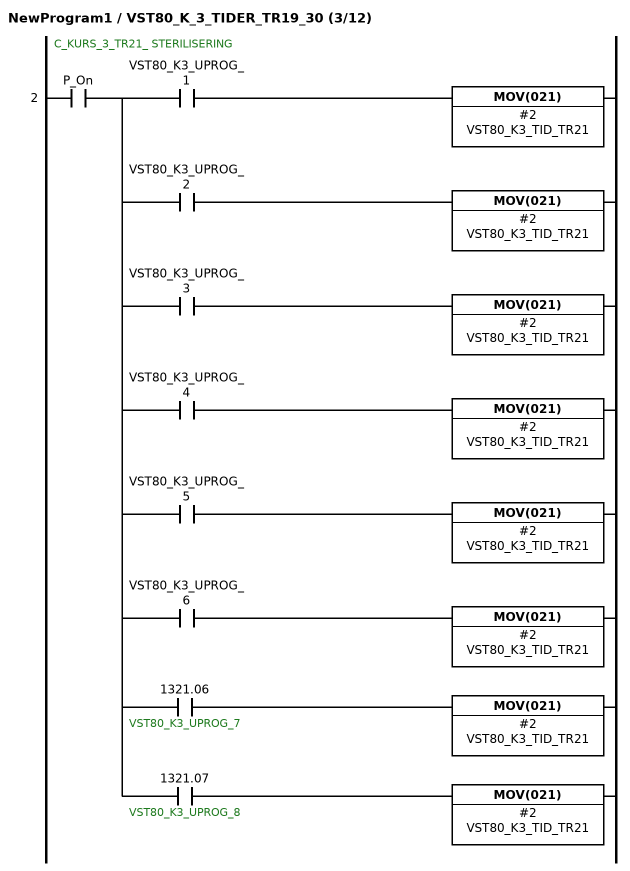
; [picture p312: NewProgram1 / VST80_K_3_TIDER_TR19_30, rungs 2-2]
; rung 2: C_KURS_3_TR21_ STERILISERING
LD P_On
OUT TR0
AND VST80_K3_UPROG_1
MOV(021) #2 VST80_K3_TID_TR21
LD TR0
AND VST80_K3_UPROG_2
MOV(021) #2 VST80_K3_TID_TR21
LD TR0
AND VST80_K3_UPROG_3
MOV(021) #2 VST80_K3_TID_TR21
LD TR0
AND VST80_K3_UPROG_4
MOV(021) #2 VST80_K3_TID_TR21
LD TR0
AND VST80_K3_UPROG_5
MOV(021) #2 VST80_K3_TID_TR21
LD TR0
AND VST80_K3_UPROG_6
MOV(021) #2 VST80_K3_TID_TR21
LD TR0
AND 1321.06  ; VST80_K3_UPROG_7
MOV(021) #2 VST80_K3_TID_TR21
LD TR0
AND 1321.07  ; VST80_K3_UPROG_8
MOV(021) #2 VST80_K3_TID_TR21

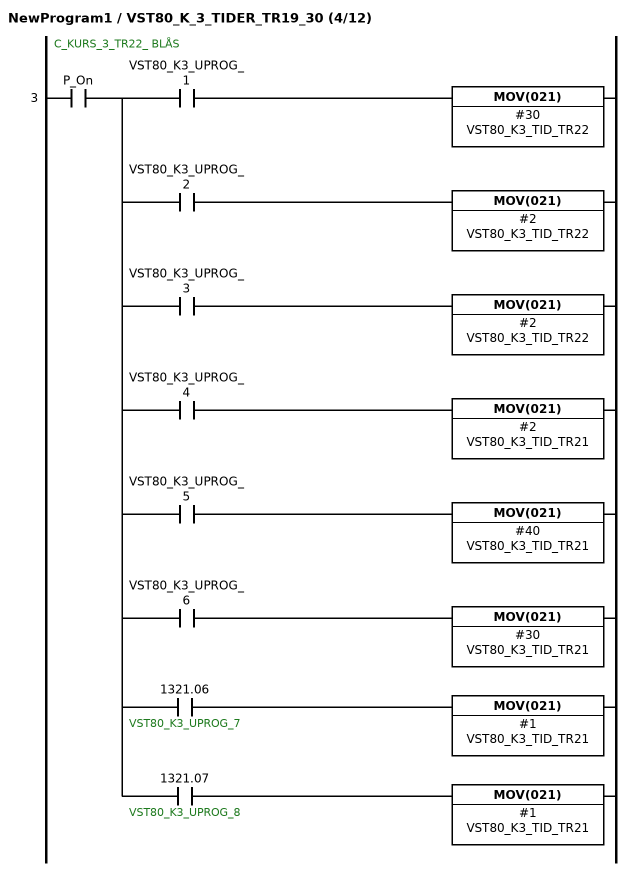
; rung 3: C_KURS_3_TR22_ BLÅS
LD P_On
OUT TR0
AND VST80_K3_UPROG_1
MOV(021) #30 VST80_K3_TID_TR22
LD TR0
AND VST80_K3_UPROG_2
MOV(021) #2 VST80_K3_TID_TR22
LD TR0
AND VST80_K3_UPROG_3
MOV(021) #2 VST80_K3_TID_TR22
LD TR0
AND VST80_K3_UPROG_4
MOV(021) #2 VST80_K3_TID_TR21
LD TR0
AND VST80_K3_UPROG_5
MOV(021) #40 VST80_K3_TID_TR21
LD TR0
AND VST80_K3_UPROG_6
MOV(021) #30 VST80_K3_TID_TR21
LD TR0
AND 1321.06  ; VST80_K3_UPROG_7
MOV(021) #1 VST80_K3_TID_TR21
LD TR0
AND 1321.07  ; VST80_K3_UPROG_8
MOV(021) #1 VST80_K3_TID_TR21

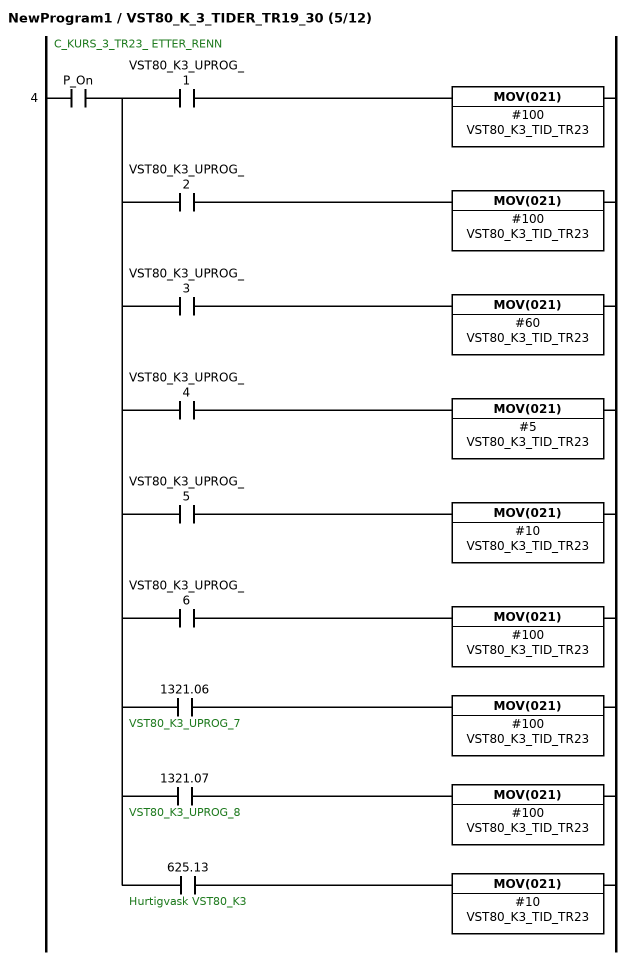
; rung 4: C_KURS_3_TR23_ ETTER_RENN
LD P_On
OUT TR0
AND VST80_K3_UPROG_1
MOV(021) #100 VST80_K3_TID_TR23
LD TR0
AND VST80_K3_UPROG_2
MOV(021) #100 VST80_K3_TID_TR23
LD TR0
AND VST80_K3_UPROG_3
MOV(021) #60 VST80_K3_TID_TR23
LD TR0
AND VST80_K3_UPROG_4
MOV(021) #5 VST80_K3_TID_TR23
LD TR0
AND VST80_K3_UPROG_5
MOV(021) #10 VST80_K3_TID_TR23
LD TR0
AND VST80_K3_UPROG_6
MOV(021) #100 VST80_K3_TID_TR23
LD TR0
AND 1321.06  ; VST80_K3_UPROG_7
MOV(021) #100 VST80_K3_TID_TR23
LD TR0
AND 1321.07  ; VST80_K3_UPROG_8
MOV(021) #100 VST80_K3_TID_TR23
LD TR0
AND 625.13  ; Hurtigvask VST80_K3
MOV(021) #10 VST80_K3_TID_TR23

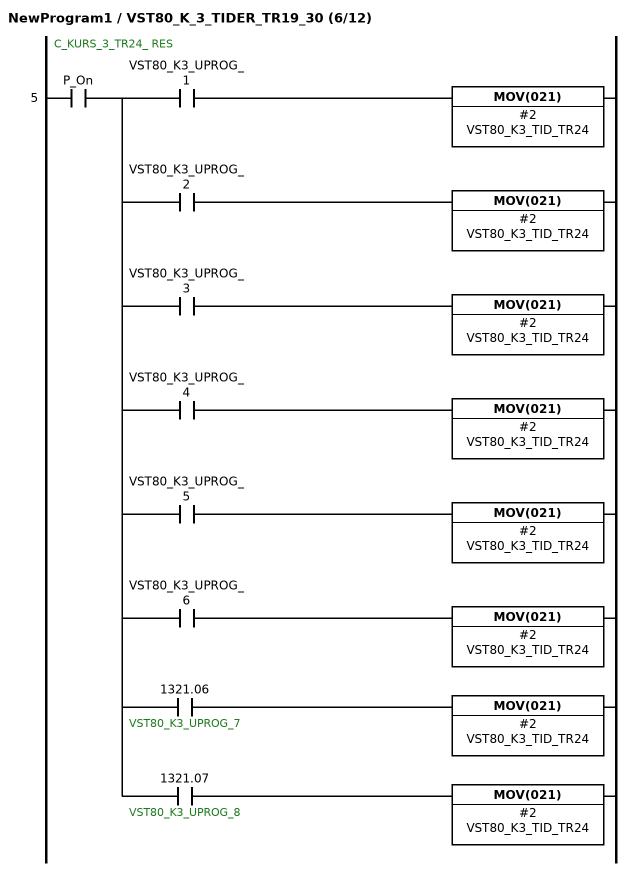
; rung 5: C_KURS_3_TR24_ RES
LD P_On
OUT TR0
AND VST80_K3_UPROG_1
MOV(021) #2 VST80_K3_TID_TR24
LD TR0
AND VST80_K3_UPROG_2
MOV(021) #2 VST80_K3_TID_TR24
LD TR0
AND VST80_K3_UPROG_3
MOV(021) #2 VST80_K3_TID_TR24
LD TR0
AND VST80_K3_UPROG_4
MOV(021) #2 VST80_K3_TID_TR24
LD TR0
AND VST80_K3_UPROG_5
MOV(021) #2 VST80_K3_TID_TR24
LD TR0
AND VST80_K3_UPROG_6
MOV(021) #2 VST80_K3_TID_TR24
LD TR0
AND 1321.06  ; VST80_K3_UPROG_7
MOV(021) #2 VST80_K3_TID_TR24
LD TR0
AND 1321.07  ; VST80_K3_UPROG_8
MOV(021) #2 VST80_K3_TID_TR24

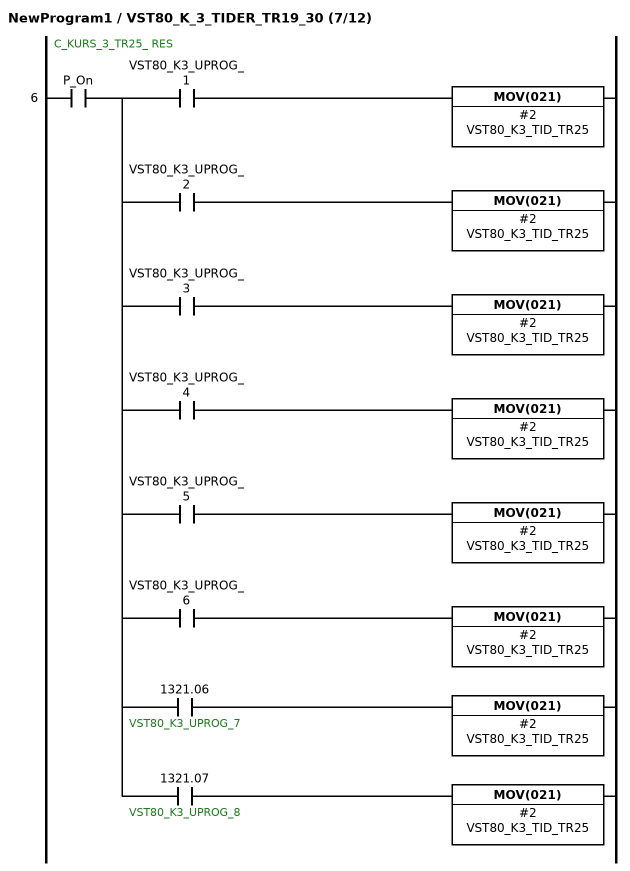
; rung 6: C_KURS_3_TR25_ RES
LD P_On
OUT TR0
AND VST80_K3_UPROG_1
MOV(021) #2 VST80_K3_TID_TR25
LD TR0
AND VST80_K3_UPROG_2
MOV(021) #2 VST80_K3_TID_TR25
LD TR0
AND VST80_K3_UPROG_3
MOV(021) #2 VST80_K3_TID_TR25
LD TR0
AND VST80_K3_UPROG_4
MOV(021) #2 VST80_K3_TID_TR25
LD TR0
AND VST80_K3_UPROG_5
MOV(021) #2 VST80_K3_TID_TR25
LD TR0
AND VST80_K3_UPROG_6
MOV(021) #2 VST80_K3_TID_TR25
LD TR0
AND 1321.06  ; VST80_K3_UPROG_7
MOV(021) #2 VST80_K3_TID_TR25
LD TR0
AND 1321.07  ; VST80_K3_UPROG_8
MOV(021) #2 VST80_K3_TID_TR25

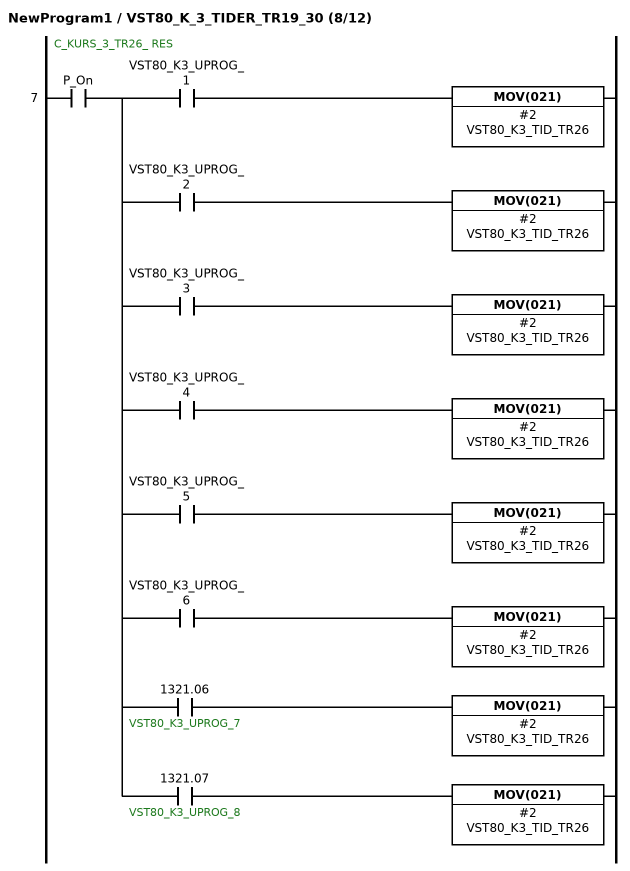
; rung 7: C_KURS_3_TR26_ RES
LD P_On
OUT TR0
AND VST80_K3_UPROG_1
MOV(021) #2 VST80_K3_TID_TR26
LD TR0
AND VST80_K3_UPROG_2
MOV(021) #2 VST80_K3_TID_TR26
LD TR0
AND VST80_K3_UPROG_3
MOV(021) #2 VST80_K3_TID_TR26
LD TR0
AND VST80_K3_UPROG_4
MOV(021) #2 VST80_K3_TID_TR26
LD TR0
AND VST80_K3_UPROG_5
MOV(021) #2 VST80_K3_TID_TR26
LD TR0
AND VST80_K3_UPROG_6
MOV(021) #2 VST80_K3_TID_TR26
LD TR0
AND 1321.06  ; VST80_K3_UPROG_7
MOV(021) #2 VST80_K3_TID_TR26
LD TR0
AND 1321.07  ; VST80_K3_UPROG_8
MOV(021) #2 VST80_K3_TID_TR26

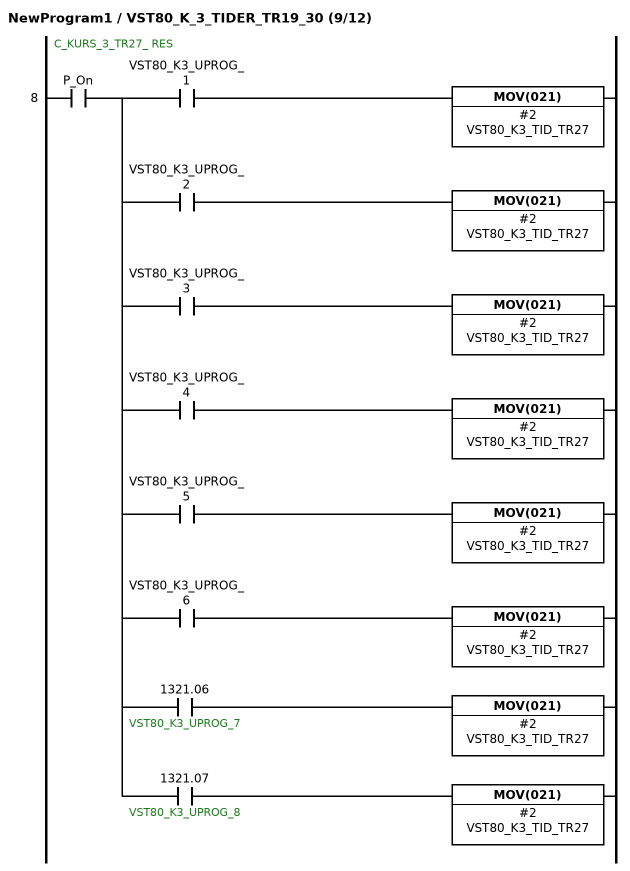
; rung 8: C_KURS_3_TR27_ RES
LD P_On
OUT TR0
AND VST80_K3_UPROG_1
MOV(021) #2 VST80_K3_TID_TR27
LD TR0
AND VST80_K3_UPROG_2
MOV(021) #2 VST80_K3_TID_TR27
LD TR0
AND VST80_K3_UPROG_3
MOV(021) #2 VST80_K3_TID_TR27
LD TR0
AND VST80_K3_UPROG_4
MOV(021) #2 VST80_K3_TID_TR27
LD TR0
AND VST80_K3_UPROG_5
MOV(021) #2 VST80_K3_TID_TR27
LD TR0
AND VST80_K3_UPROG_6
MOV(021) #2 VST80_K3_TID_TR27
LD TR0
AND 1321.06  ; VST80_K3_UPROG_7
MOV(021) #2 VST80_K3_TID_TR27
LD TR0
AND 1321.07  ; VST80_K3_UPROG_8
MOV(021) #2 VST80_K3_TID_TR27

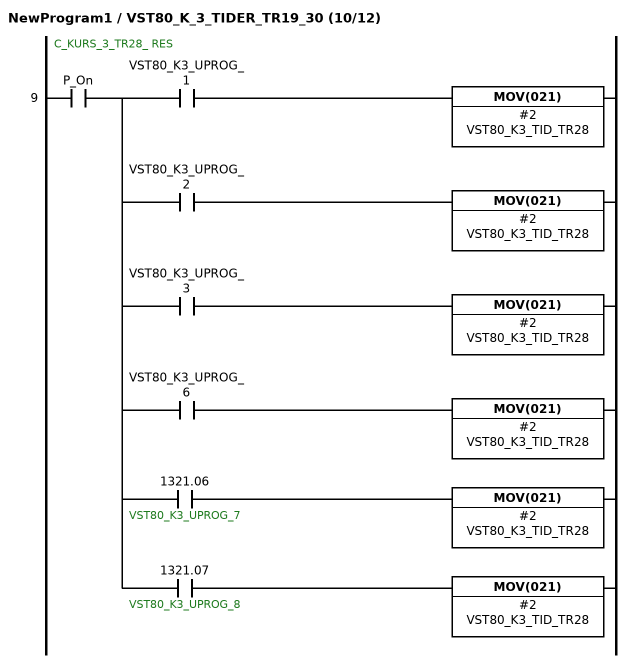
; rung 9: C_KURS_3_TR28_ RES
LD P_On
OUT TR0
AND VST80_K3_UPROG_1
MOV(021) #2 VST80_K3_TID_TR28
LD TR0
AND VST80_K3_UPROG_2
MOV(021) #2 VST80_K3_TID_TR28
LD TR0
AND VST80_K3_UPROG_3
MOV(021) #2 VST80_K3_TID_TR28
LD TR0
AND VST80_K3_UPROG_6
MOV(021) #2 VST80_K3_TID_TR28
LD TR0
AND 1321.06  ; VST80_K3_UPROG_7
MOV(021) #2 VST80_K3_TID_TR28
LD TR0
AND 1321.07  ; VST80_K3_UPROG_8
MOV(021) #2 VST80_K3_TID_TR28

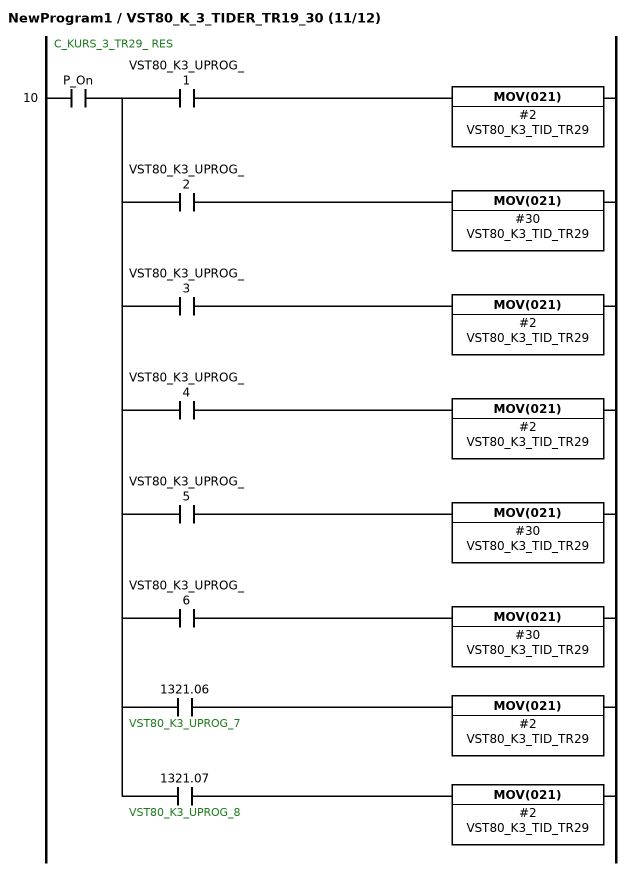
; rung 10: C_KURS_3_TR29_ RES
LD P_On
OUT TR0
AND VST80_K3_UPROG_1
MOV(021) #2 VST80_K3_TID_TR29
LD TR0
AND VST80_K3_UPROG_2
MOV(021) #30 VST80_K3_TID_TR29
LD TR0
AND VST80_K3_UPROG_3
MOV(021) #2 VST80_K3_TID_TR29
LD TR0
AND VST80_K3_UPROG_4
MOV(021) #2 VST80_K3_TID_TR29
LD TR0
AND VST80_K3_UPROG_5
MOV(021) #30 VST80_K3_TID_TR29
LD TR0
AND VST80_K3_UPROG_6
MOV(021) #30 VST80_K3_TID_TR29
LD TR0
AND 1321.06  ; VST80_K3_UPROG_7
MOV(021) #2 VST80_K3_TID_TR29
LD TR0
AND 1321.07  ; VST80_K3_UPROG_8
MOV(021) #2 VST80_K3_TID_TR29

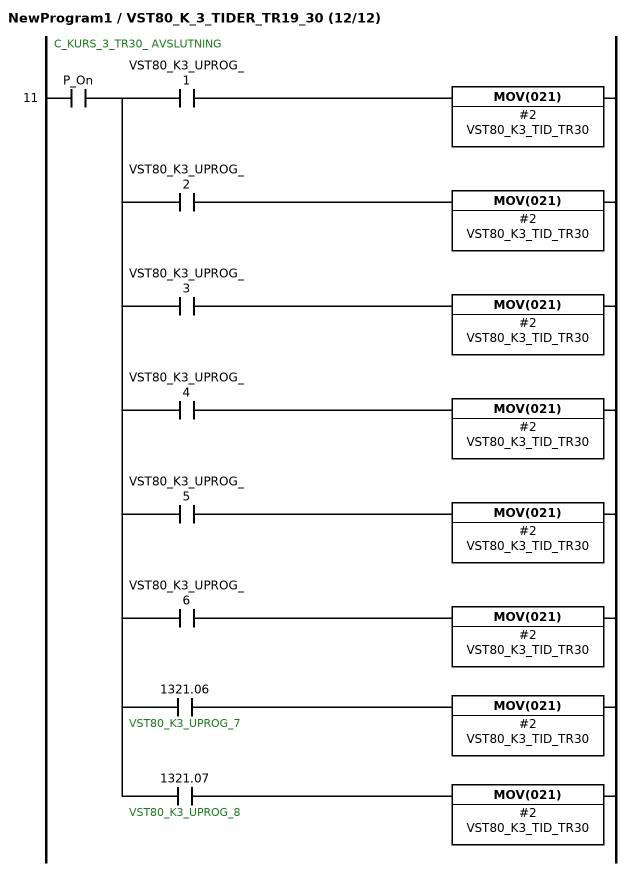
; rung 11: C_KURS_3_TR30_ AVSLUTNING
LD P_On
OUT TR0
AND VST80_K3_UPROG_1
MOV(021) #2 VST80_K3_TID_TR30
LD TR0
AND VST80_K3_UPROG_2
MOV(021) #2 VST80_K3_TID_TR30
LD TR0
AND VST80_K3_UPROG_3
MOV(021) #2 VST80_K3_TID_TR30
LD TR0
AND VST80_K3_UPROG_4
MOV(021) #2 VST80_K3_TID_TR30
LD TR0
AND VST80_K3_UPROG_5
MOV(021) #2 VST80_K3_TID_TR30
LD TR0
AND VST80_K3_UPROG_6
MOV(021) #2 VST80_K3_TID_TR30
LD TR0
AND 1321.06  ; VST80_K3_UPROG_7
MOV(021) #2 VST80_K3_TID_TR30
LD TR0
AND 1321.07  ; VST80_K3_UPROG_8
MOV(021) #2 VST80_K3_TID_TR30

### Section VST80_K3_TRINN
; Vaskeprogrammet består av 30. hovedtrinn. / Funksjonsbenstabell: 975100-BL48

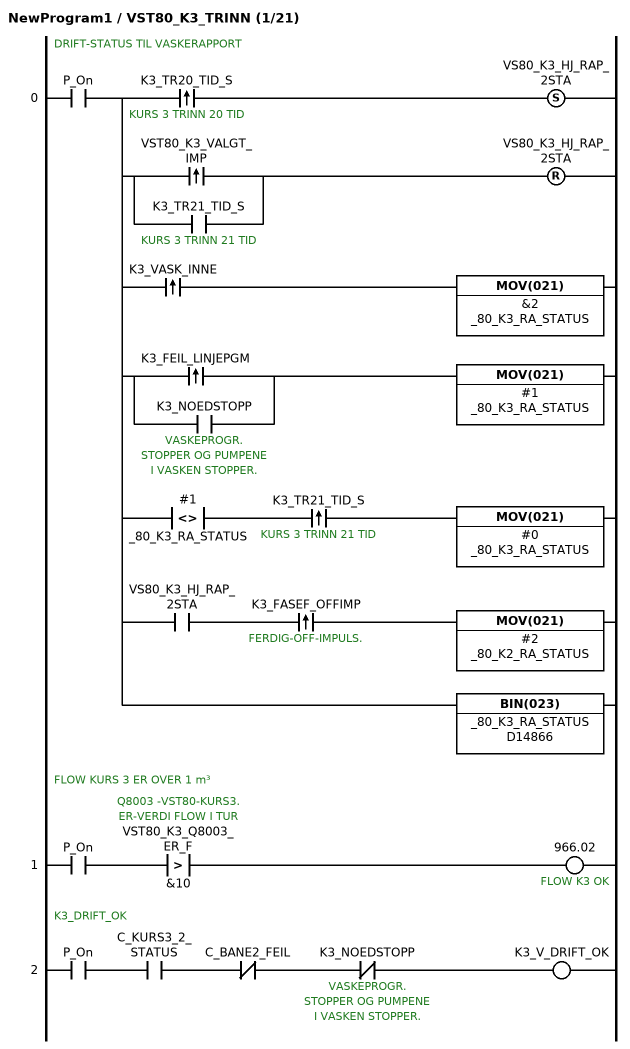
; rung 0: DRIFT-STATUS TIL VASKERAPPORT
LD P_On
OUT TR0
@AND K3_TR20_TID_S  ; KURS 3 TRINN 20 TID
SET VS80_K3_HJ_RAP_2STA
LD TR0
@LD VST80_K3_VALGT_IMP
OR K3_TR21_TID_S  ; KURS 3 TRINN 21 TID
ANDLD
RSET VS80_K3_HJ_RAP_2STA
LD TR0
@AND K3_VASK_INNE
MOV(021) &2 _80_K3_RA_STATUS
LD TR0
@LD K3_FEIL_LINJEPGM
OR K3_NOEDSTOPP  ; VASKEPROGR. STOPPER OG PUMPENE I VASKEN STOPPER.
ANDLD
MOV(021) #1 _80_K3_RA_STATUS
LD TR0
AND<>(305) #1 _80_K3_RA_STATUS
@AND K3_TR21_TID_S  ; KURS 3 TRINN 21 TID
MOV(021) #0 _80_K3_RA_STATUS
LD TR0
AND VS80_K3_HJ_RAP_2STA
@AND K3_FASEF_OFFIMP  ; FERDIG-OFF-IMPULS.
MOV(021) #2 _80_K2_RA_STATUS
LD TR0
BIN(023) _80_K3_RA_STATUS D14866
; rung 1: FLOW KURS 3 ER OVER 1 m³
LD P_On
AND>(320) VST80_K3_Q8003_ER_F &10  ; Q8003 -VST80-KURS3. ER-VERDI FLOW I TUR
OUT 966.02  ; FLOW K3 OK
; rung 2: K3_DRIFT_OK
LD P_On
AND C_KURS3_2_STATUS
ANDNOT C_BANE2_FEIL
ANDNOT K3_NOEDSTOPP  ; VASKEPROGR. STOPPER OG PUMPENE I VASKEN STOPPER.
OUT K3_V_DRIFT_OK

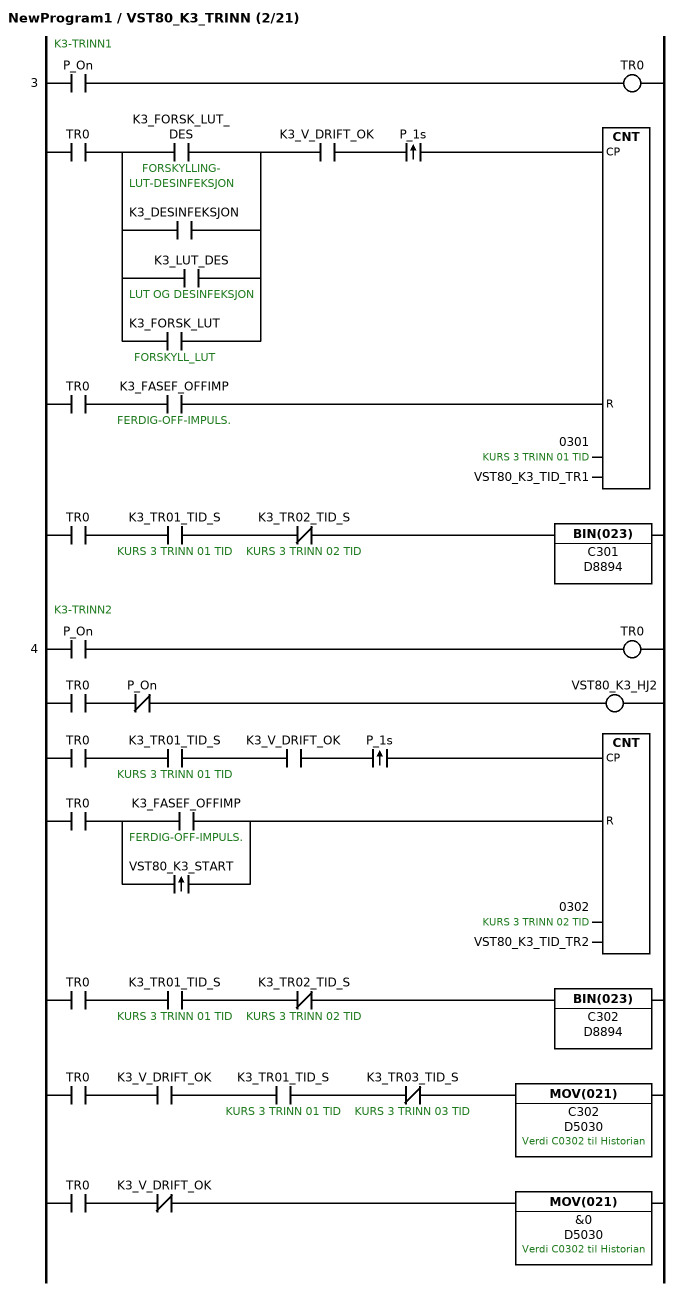
; rung 3: K3-TRINN1
LD P_On
OUT TR0
LD K3_FORSK_LUT_DES  ; FORSKYLLING- LUT-DESINFEKSJON
OR K3_DESINFEKSJON
OR K3_LUT_DES  ; LUT OG DESINFEKSJON
OR K3_FORSK_LUT  ; FORSKYLL_LUT
ANDLD
AND K3_V_DRIFT_OK
@AND P_1s
LD TR0
AND K3_FASEF_OFFIMP  ; FERDIG-OFF-IMPULS.
CNT 0301 VST80_K3_TID_TR1  ; KURS 3 TRINN 01 TID
LD TR0
AND K3_TR01_TID_S  ; KURS 3 TRINN 01 TID
ANDNOT K3_TR02_TID_S  ; KURS 3 TRINN 02 TID
BIN(023) C301 D8894
; rung 4: K3-TRINN2
LD P_On
OUT TR0
ANDNOT P_On
OUT VST80_K3_HJ2
LD TR0
AND K3_TR01_TID_S  ; KURS 3 TRINN 01 TID
AND K3_V_DRIFT_OK
@AND P_1s
LD TR0
LD K3_FASEF_OFFIMP  ; FERDIG-OFF-IMPULS.
@OR VST80_K3_START
ANDLD
CNT 0302 VST80_K3_TID_TR2  ; KURS 3 TRINN 02 TID
LD TR0
AND K3_TR01_TID_S  ; KURS 3 TRINN 01 TID
ANDNOT K3_TR02_TID_S  ; KURS 3 TRINN 02 TID
BIN(023) C302 D8894
LD TR0
AND K3_V_DRIFT_OK
AND K3_TR01_TID_S  ; KURS 3 TRINN 01 TID
ANDNOT K3_TR03_TID_S  ; KURS 3 TRINN 03 TID
MOV(021) C302 D5030  ; Verdi C0302 til Historian
LD TR0
ANDNOT K3_V_DRIFT_OK
MOV(021) &0 D5030  ; Verdi C0302 til Historian

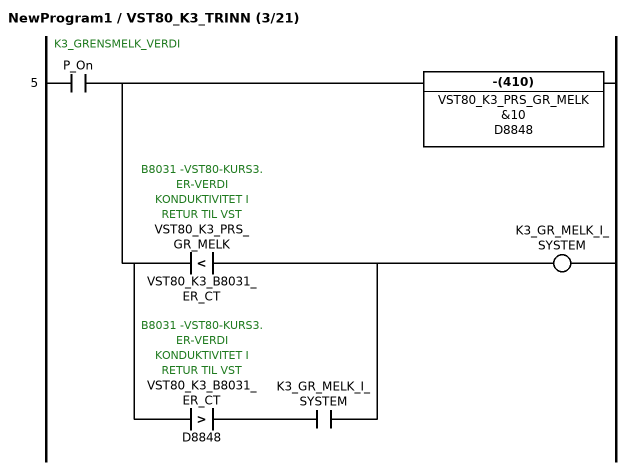
; rung 5: K3_GRENSMELK_VERDI
LD P_On
-(410) VST80_K3_PRS_GR_MELK &10 D8848
LD<(310) VST80_K3_PRS_GR_MELK VST80_K3_B8031_ER_CT  ; B8031 -VST80-KURS3. ER-VERDI KONDUKTIVITET I RETUR TIL VST
LD>(320) VST80_K3_B8031_ER_CT D8848  ; B8031 -VST80-KURS3. ER-VERDI KONDUKTIVITET I RETUR TIL VST
AND K3_GR_MELK_I_SYSTEM
ORLD
ANDLD
OUT K3_GR_MELK_I_SYSTEM

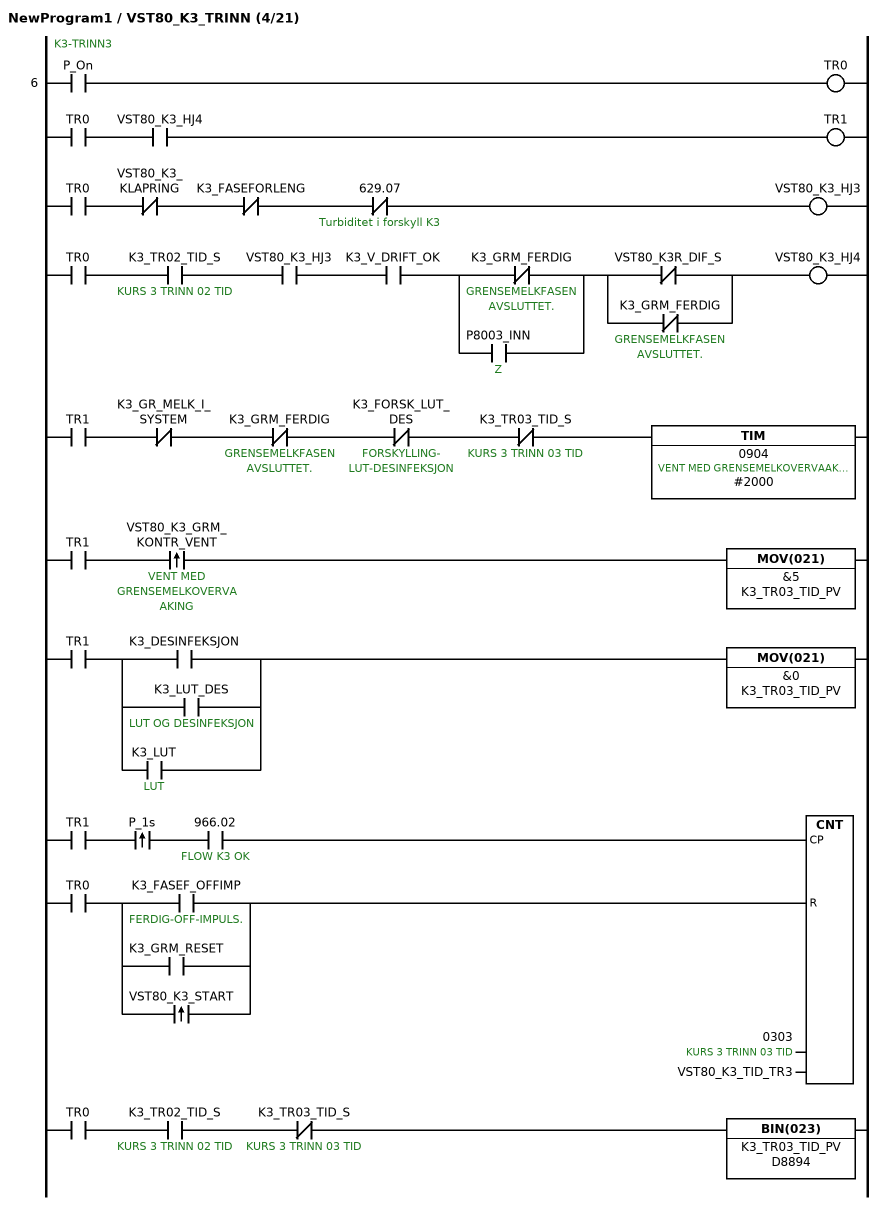
; rung 6: K3-TRINN3
LD P_On
OUT TR0
ANDNOT VST80_K3_KLAPRING
ANDNOT K3_FASEFORLENG
ANDNOT 629.07  ; Turbiditet i forskyll K3
OUT VST80_K3_HJ3
LD TR0
AND K3_TR02_TID_S  ; KURS 3 TRINN 02 TID
AND VST80_K3_HJ3
AND K3_V_DRIFT_OK
LDNOT K3_GRM_FERDIG  ; GRENSEMELKFASEN AVSLUTTET.
OR P8003_INN  ; Z
ANDLD
LDNOT VST80_K3R_DIF_S
ORNOT K3_GRM_FERDIG  ; GRENSEMELKFASEN AVSLUTTET.
ANDLD
OUT VST80_K3_HJ4
LD TR0
AND VST80_K3_HJ4
OUT TR1
ANDNOT K3_GR_MELK_I_SYSTEM
ANDNOT K3_GRM_FERDIG  ; GRENSEMELKFASEN AVSLUTTET.
ANDNOT K3_FORSK_LUT_DES  ; FORSKYLLING- LUT-DESINFEKSJON
ANDNOT K3_TR03_TID_S  ; KURS 3 TRINN 03 TID
TIM 0904 #2000  ; VENT MED GRENSEMELKOVERVAAKING
LD TR1
@AND VST80_K3_GRM_KONTR_VENT  ; VENT MED GRENSEMELKOVERVAAKING
MOV(021) &5 K3_TR03_TID_PV
LD TR1
LD K3_DESINFEKSJON
OR K3_LUT_DES  ; LUT OG DESINFEKSJON
OR K3_LUT  ; LUT
ANDLD
MOV(021) &0 K3_TR03_TID_PV
LD TR1
@AND P_1s
AND 966.02  ; FLOW K3 OK
LD TR0
LD K3_FASEF_OFFIMP  ; FERDIG-OFF-IMPULS.
OR K3_GRM_RESET
@OR VST80_K3_START
ANDLD
CNT 0303 VST80_K3_TID_TR3  ; KURS 3 TRINN 03 TID
LD TR0
AND K3_TR02_TID_S  ; KURS 3 TRINN 02 TID
ANDNOT K3_TR03_TID_S  ; KURS 3 TRINN 03 TID
BIN(023) K3_TR03_TID_PV D8894

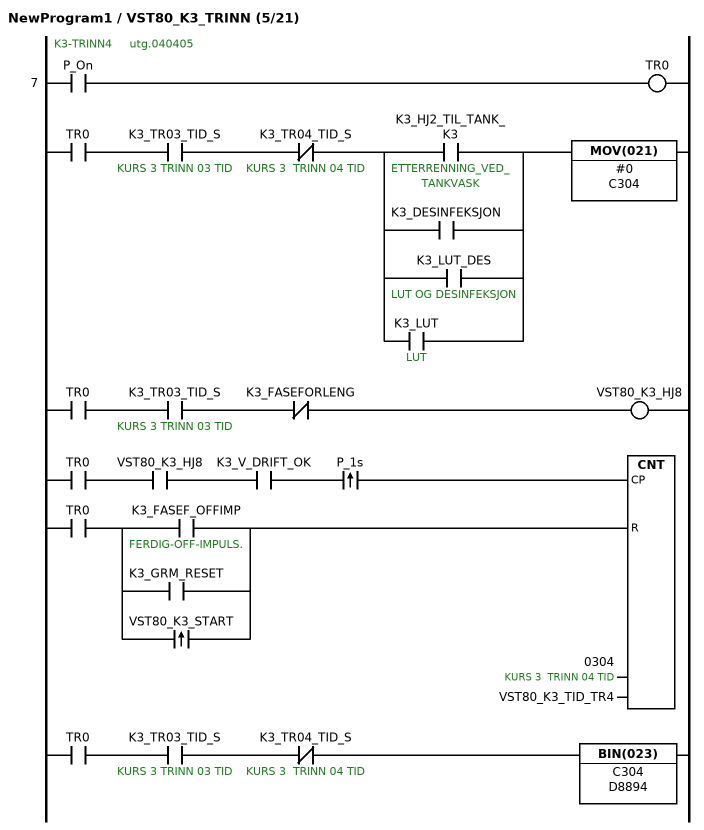
; rung 7: K3-TRINN4     utg.040405
LD P_On
OUT TR0
AND K3_TR03_TID_S  ; KURS 3 TRINN 03 TID
ANDNOT K3_TR04_TID_S  ; KURS 3  TRINN 04 TID
LD K3_HJ2_TIL_TANK_K3  ; ETTERRENNING_VED_TANKVASK
OR K3_DESINFEKSJON
OR K3_LUT_DES  ; LUT OG DESINFEKSJON
OR K3_LUT  ; LUT
ANDLD
MOV(021) #0 C304
LD TR0
AND K3_TR03_TID_S  ; KURS 3 TRINN 03 TID
ANDNOT K3_FASEFORLENG
OUT VST80_K3_HJ8
LD TR0
AND VST80_K3_HJ8
AND K3_V_DRIFT_OK
@AND P_1s
LD TR0
LD K3_FASEF_OFFIMP  ; FERDIG-OFF-IMPULS.
OR K3_GRM_RESET
@OR VST80_K3_START
ANDLD
CNT 0304 VST80_K3_TID_TR4  ; KURS 3  TRINN 04 TID
LD TR0
AND K3_TR03_TID_S  ; KURS 3 TRINN 03 TID
ANDNOT K3_TR04_TID_S  ; KURS 3  TRINN 04 TID
BIN(023) C304 D8894

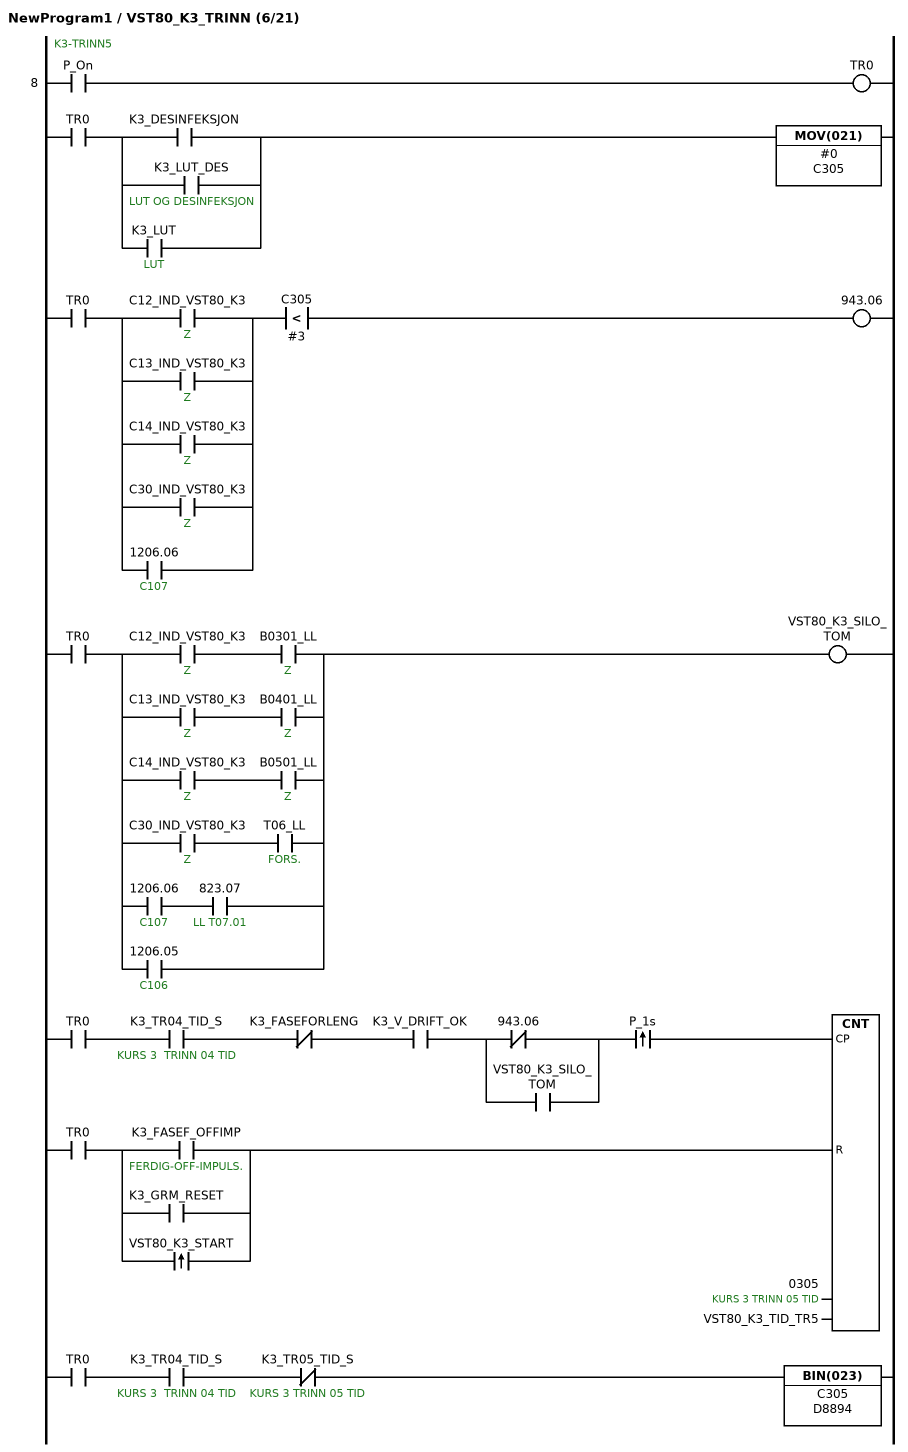
; rung 8: K3-TRINN5
LD P_On
OUT TR0
LD K3_DESINFEKSJON
OR K3_LUT_DES  ; LUT OG DESINFEKSJON
OR K3_LUT  ; LUT
ANDLD
MOV(021) #0 C305
LD TR0
LD C12_IND_VST80_K3  ; Z
OR C13_IND_VST80_K3  ; Z
OR C14_IND_VST80_K3  ; Z
OR C30_IND_VST80_K3  ; Z
OR 1206.06  ; C107
ANDLD
AND<(310) C305 #3
OUT 943.06
LD TR0
LD C12_IND_VST80_K3  ; Z
AND B0301_LL  ; Z
LD C13_IND_VST80_K3  ; Z
AND B0401_LL  ; Z
ORLD
LD C14_IND_VST80_K3  ; Z
AND B0501_LL  ; Z
ORLD
LD C30_IND_VST80_K3  ; Z
AND T06_LL  ; FORS.
ORLD
LD 1206.06  ; C107
AND 823.07  ; LL T07.01
ORLD
OR 1206.05  ; C106
ANDLD
OUT VST80_K3_SILO_TOM
LD TR0
AND K3_TR04_TID_S  ; KURS 3  TRINN 04 TID
ANDNOT K3_FASEFORLENG
AND K3_V_DRIFT_OK
LDNOT 943.06
OR VST80_K3_SILO_TOM
ANDLD
@AND P_1s
LD TR0
LD K3_FASEF_OFFIMP  ; FERDIG-OFF-IMPULS.
OR K3_GRM_RESET
@OR VST80_K3_START
ANDLD
CNT 0305 VST80_K3_TID_TR5  ; KURS 3 TRINN 05 TID
LD TR0
AND K3_TR04_TID_S  ; KURS 3  TRINN 04 TID
ANDNOT K3_TR05_TID_S  ; KURS 3 TRINN 05 TID
BIN(023) C305 D8894

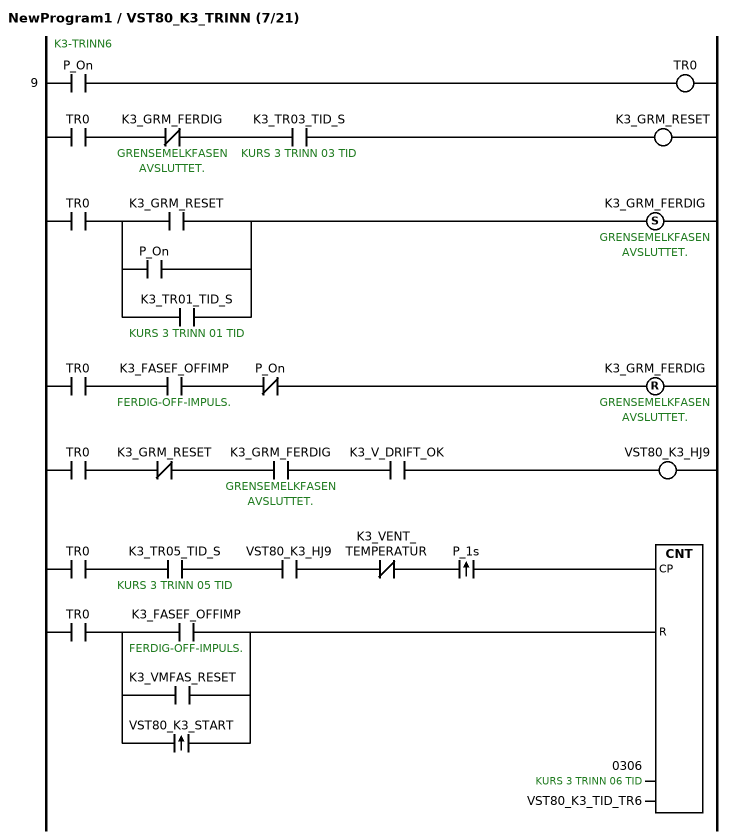
; rung 9: K3-TRINN6
LD P_On
OUT TR0
ANDNOT K3_GRM_FERDIG  ; GRENSEMELKFASEN AVSLUTTET.
AND K3_TR03_TID_S  ; KURS 3 TRINN 03 TID
OUT K3_GRM_RESET
LD TR0
LD K3_GRM_RESET
OR P_On
OR K3_TR01_TID_S  ; KURS 3 TRINN 01 TID
ANDLD
SET K3_GRM_FERDIG  ; GRENSEMELKFASEN AVSLUTTET.
LD TR0
AND K3_FASEF_OFFIMP  ; FERDIG-OFF-IMPULS.
ANDNOT P_On
RSET K3_GRM_FERDIG  ; GRENSEMELKFASEN AVSLUTTET.
LD TR0
ANDNOT K3_GRM_RESET
AND K3_GRM_FERDIG  ; GRENSEMELKFASEN AVSLUTTET.
AND K3_V_DRIFT_OK
OUT VST80_K3_HJ9
LD TR0
AND K3_TR05_TID_S  ; KURS 3 TRINN 05 TID
AND VST80_K3_HJ9
ANDNOT K3_VENT_TEMPERATUR
@AND P_1s
LD TR0
LD K3_FASEF_OFFIMP  ; FERDIG-OFF-IMPULS.
OR K3_VMFAS_RESET
@OR VST80_K3_START
ANDLD
CNT 0306 VST80_K3_TID_TR6  ; KURS 3 TRINN 06 TID

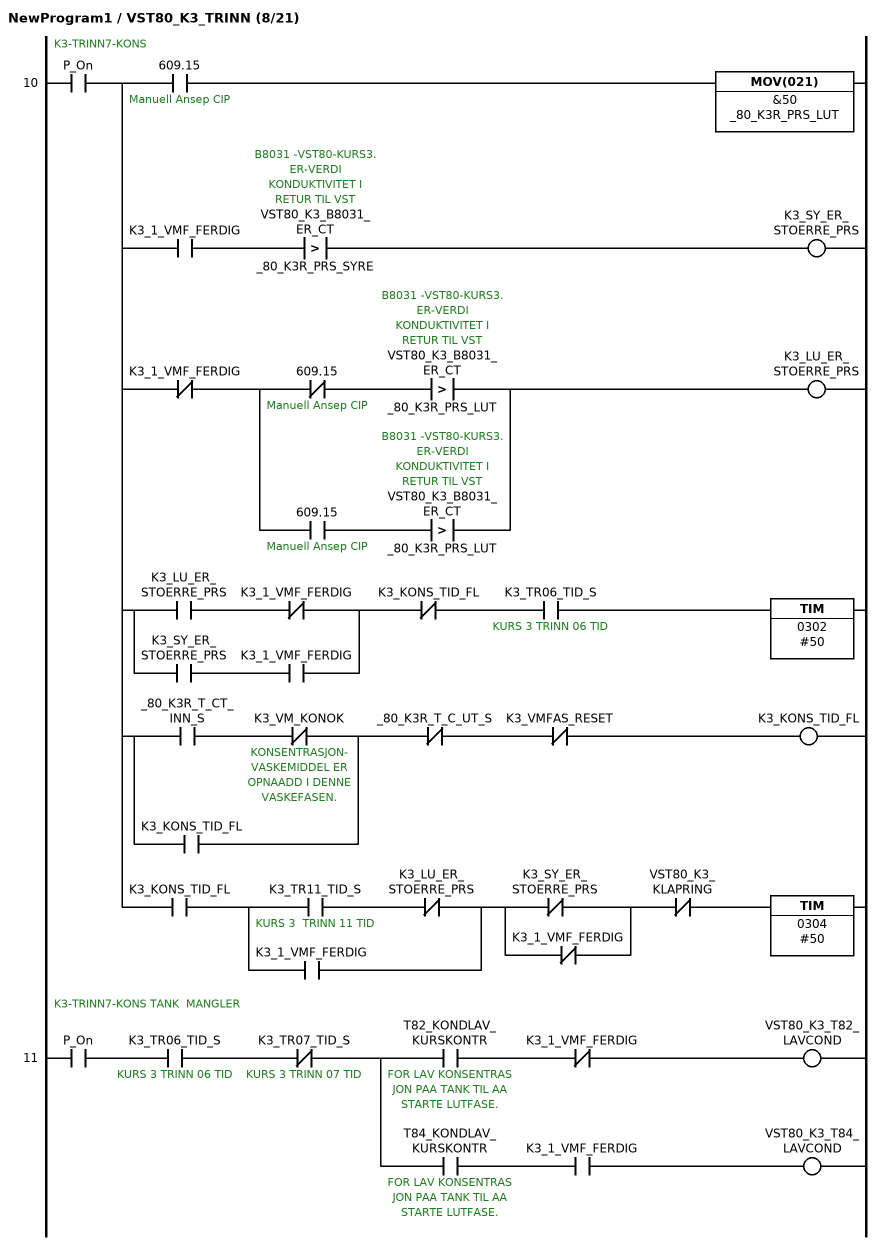
; rung 10: K3-TRINN7-KONS
LD P_On
OUT TR0
AND 609.15  ; Manuell Ansep CIP
MOV(021) &50 _80_K3R_PRS_LUT
LD TR0
AND K3_1_VMF_FERDIG
AND>(320) VST80_K3_B8031_ER_CT _80_K3R_PRS_SYRE  ; B8031 -VST80-KURS3. ER-VERDI KONDUKTIVITET I RETUR TIL VST
OUT K3_SY_ER_STOERRE_PRS
LD TR0
ANDNOT K3_1_VMF_FERDIG
LDNOT 609.15  ; Manuell Ansep CIP
AND>(320) VST80_K3_B8031_ER_CT _80_K3R_PRS_LUT  ; B8031 -VST80-KURS3. ER-VERDI KONDUKTIVITET I RETUR TIL VST
LD 609.15  ; Manuell Ansep CIP
AND>(320) VST80_K3_B8031_ER_CT _80_K3R_PRS_LUT  ; B8031 -VST80-KURS3. ER-VERDI KONDUKTIVITET I RETUR TIL VST
ORLD
ANDLD
OUT K3_LU_ER_STOERRE_PRS
LD TR0
LD K3_LU_ER_STOERRE_PRS
ANDNOT K3_1_VMF_FERDIG
LD K3_SY_ER_STOERRE_PRS
AND K3_1_VMF_FERDIG
ORLD
ANDLD
ANDNOT K3_KONS_TID_FL
AND K3_TR06_TID_S  ; KURS 3 TRINN 06 TID
TIM 0302 #50
LD TR0
LD _80_K3R_T_CT_INN_S
ANDNOT K3_VM_KONOK  ; KONSENTRASJON-VASKEMIDDEL ER OPNAADD I DENNE VASKEFASEN.
OR K3_KONS_TID_FL
ANDLD
ANDNOT _80_K3R_T_C_UT_S
ANDNOT K3_VMFAS_RESET
OUT K3_KONS_TID_FL
LD TR0
AND K3_KONS_TID_FL
LD K3_TR11_TID_S  ; KURS 3  TRINN 11 TID
ANDNOT K3_LU_ER_STOERRE_PRS
OR K3_1_VMF_FERDIG
ANDLD
LDNOT K3_SY_ER_STOERRE_PRS
ORNOT K3_1_VMF_FERDIG
ANDLD
ANDNOT VST80_K3_KLAPRING
TIM 0304 #50
; rung 11: K3-TRINN7-KONS TANK  MANGLER
LD P_On
AND K3_TR06_TID_S  ; KURS 3 TRINN 06 TID
ANDNOT K3_TR07_TID_S  ; KURS 3 TRINN 07 TID
OUT TR0
AND T82_KONDLAV_KURSKONTR  ; FOR LAV KONSENTRASJON PAA TANK TIL AA STARTE LUTFASE.
ANDNOT K3_1_VMF_FERDIG
OUT VST80_K3_T82_LAVCOND
LD TR0
AND T84_KONDLAV_KURSKONTR  ; FOR LAV KONSENTRASJON PAA TANK TIL AA STARTE LUTFASE.
AND K3_1_VMF_FERDIG
OUT VST80_K3_T84_LAVCOND

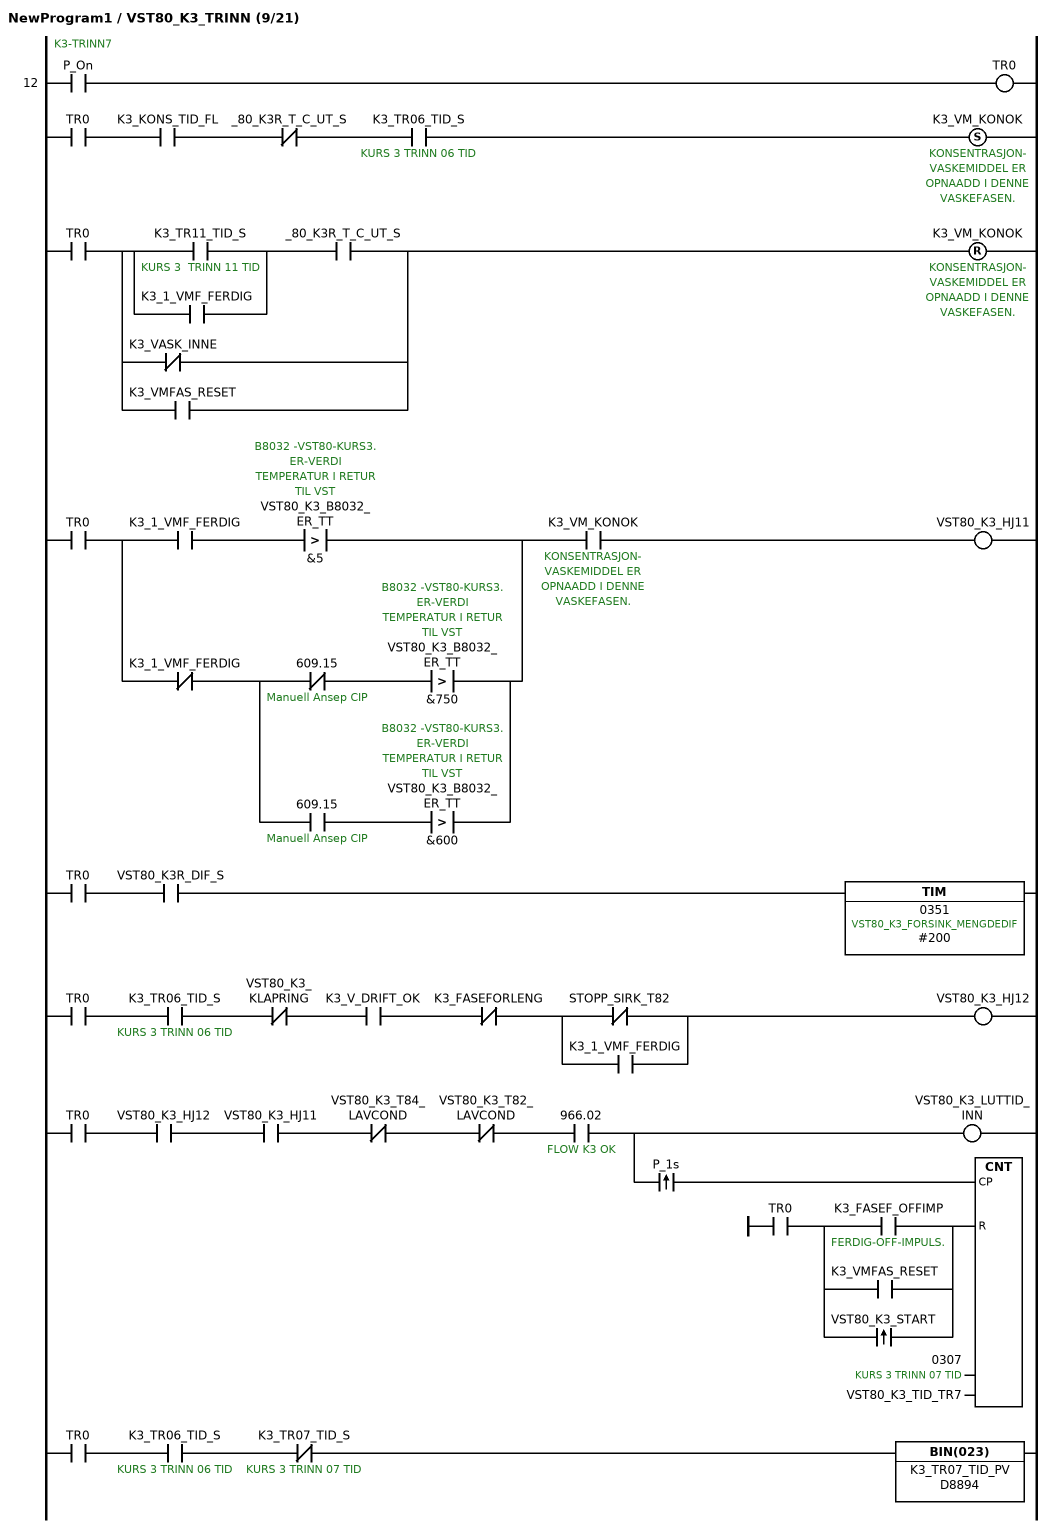
; rung 12: K3-TRINN7
LD P_On
OUT TR0
AND K3_KONS_TID_FL
ANDNOT _80_K3R_T_C_UT_S
AND K3_TR06_TID_S  ; KURS 3 TRINN 06 TID
SET K3_VM_KONOK  ; KONSENTRASJON-VASKEMIDDEL ER OPNAADD I DENNE VASKEFASEN.
LD TR0
LD K3_TR11_TID_S  ; KURS 3  TRINN 11 TID
OR K3_1_VMF_FERDIG
AND _80_K3R_T_C_UT_S
ORNOT K3_VASK_INNE
OR K3_VMFAS_RESET
ANDLD
RSET K3_VM_KONOK  ; KONSENTRASJON-VASKEMIDDEL ER OPNAADD I DENNE VASKEFASEN.
LD TR0
LD K3_1_VMF_FERDIG
AND>(320) VST80_K3_B8032_ER_TT &5  ; B8032 -VST80-KURS3. ER-VERDI TEMPERATUR I RETUR TIL VST
LDNOT K3_1_VMF_FERDIG
LDNOT 609.15  ; Manuell Ansep CIP
AND>(320) VST80_K3_B8032_ER_TT &750  ; B8032 -VST80-KURS3. ER-VERDI TEMPERATUR I RETUR TIL VST
LD 609.15  ; Manuell Ansep CIP
AND>(320) VST80_K3_B8032_ER_TT &600  ; B8032 -VST80-KURS3. ER-VERDI TEMPERATUR I RETUR TIL VST
ORLD
ANDLD
ORLD
ANDLD
AND K3_VM_KONOK  ; KONSENTRASJON-VASKEMIDDEL ER OPNAADD I DENNE VASKEFASEN.
OUT VST80_K3_HJ11
LD TR0
AND VST80_K3R_DIF_S
TIM 0351 #200  ; VST80_K3_FORSINK_MENGDEDIF
LD TR0
AND K3_TR06_TID_S  ; KURS 3 TRINN 06 TID
ANDNOT VST80_K3_KLAPRING
AND K3_V_DRIFT_OK
ANDNOT K3_FASEFORLENG
LDNOT STOPP_SIRK_T82
OR K3_1_VMF_FERDIG
ANDLD
OUT VST80_K3_HJ12
LD TR0
AND VST80_K3_HJ12
AND VST80_K3_HJ11
ANDNOT VST80_K3_T84_LAVCOND
ANDNOT VST80_K3_T82_LAVCOND
AND 966.02  ; FLOW K3 OK
OUT VST80_K3_LUTTID_INN
@AND P_1s
LD TR0
LD K3_FASEF_OFFIMP  ; FERDIG-OFF-IMPULS.
OR K3_VMFAS_RESET
@OR VST80_K3_START
ANDLD
CNT 0307 VST80_K3_TID_TR7  ; KURS 3 TRINN 07 TID
LD TR0
AND K3_TR06_TID_S  ; KURS 3 TRINN 06 TID
ANDNOT K3_TR07_TID_S  ; KURS 3 TRINN 07 TID
BIN(023) K3_TR07_TID_PV D8894

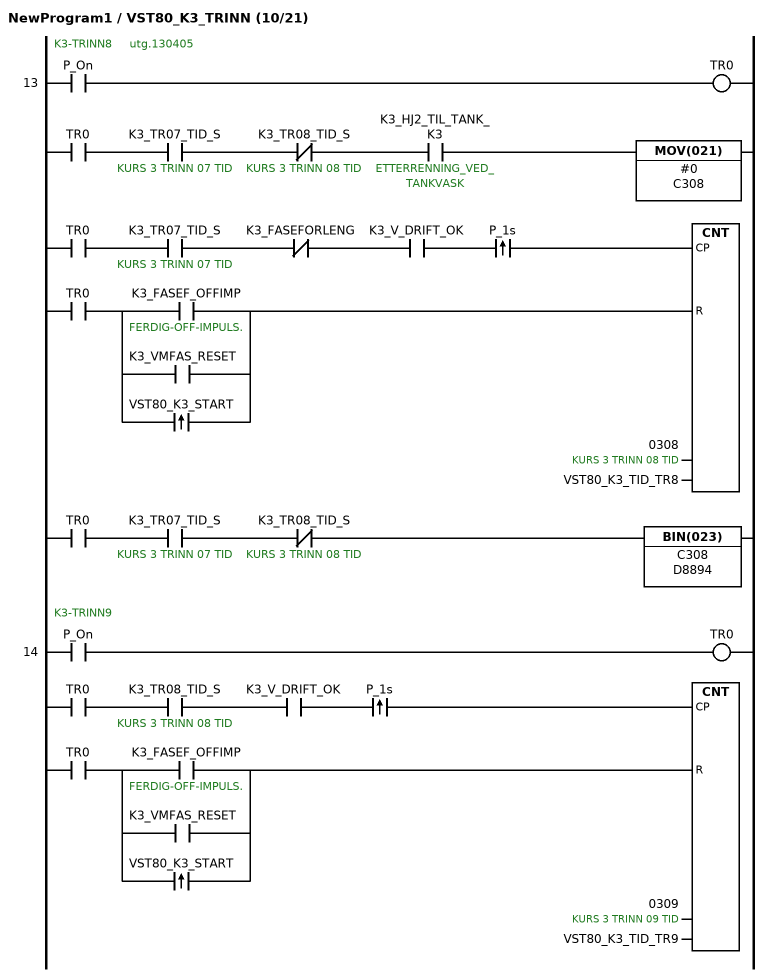
; rung 13: K3-TRINN8     utg.130405
LD P_On
OUT TR0
AND K3_TR07_TID_S  ; KURS 3 TRINN 07 TID
ANDNOT K3_TR08_TID_S  ; KURS 3 TRINN 08 TID
AND K3_HJ2_TIL_TANK_K3  ; ETTERRENNING_VED_TANKVASK
MOV(021) #0 C308
LD TR0
AND K3_TR07_TID_S  ; KURS 3 TRINN 07 TID
ANDNOT K3_FASEFORLENG
AND K3_V_DRIFT_OK
@AND P_1s
LD TR0
LD K3_FASEF_OFFIMP  ; FERDIG-OFF-IMPULS.
OR K3_VMFAS_RESET
@OR VST80_K3_START
ANDLD
CNT 0308 VST80_K3_TID_TR8  ; KURS 3 TRINN 08 TID
LD TR0
AND K3_TR07_TID_S  ; KURS 3 TRINN 07 TID
ANDNOT K3_TR08_TID_S  ; KURS 3 TRINN 08 TID
BIN(023) C308 D8894
; rung 14: K3-TRINN9
LD P_On
OUT TR0
AND K3_TR08_TID_S  ; KURS 3 TRINN 08 TID
AND K3_V_DRIFT_OK
@AND P_1s
LD TR0
LD K3_FASEF_OFFIMP  ; FERDIG-OFF-IMPULS.
OR K3_VMFAS_RESET
@OR VST80_K3_START
ANDLD
CNT 0309 VST80_K3_TID_TR9  ; KURS 3 TRINN 09 TID

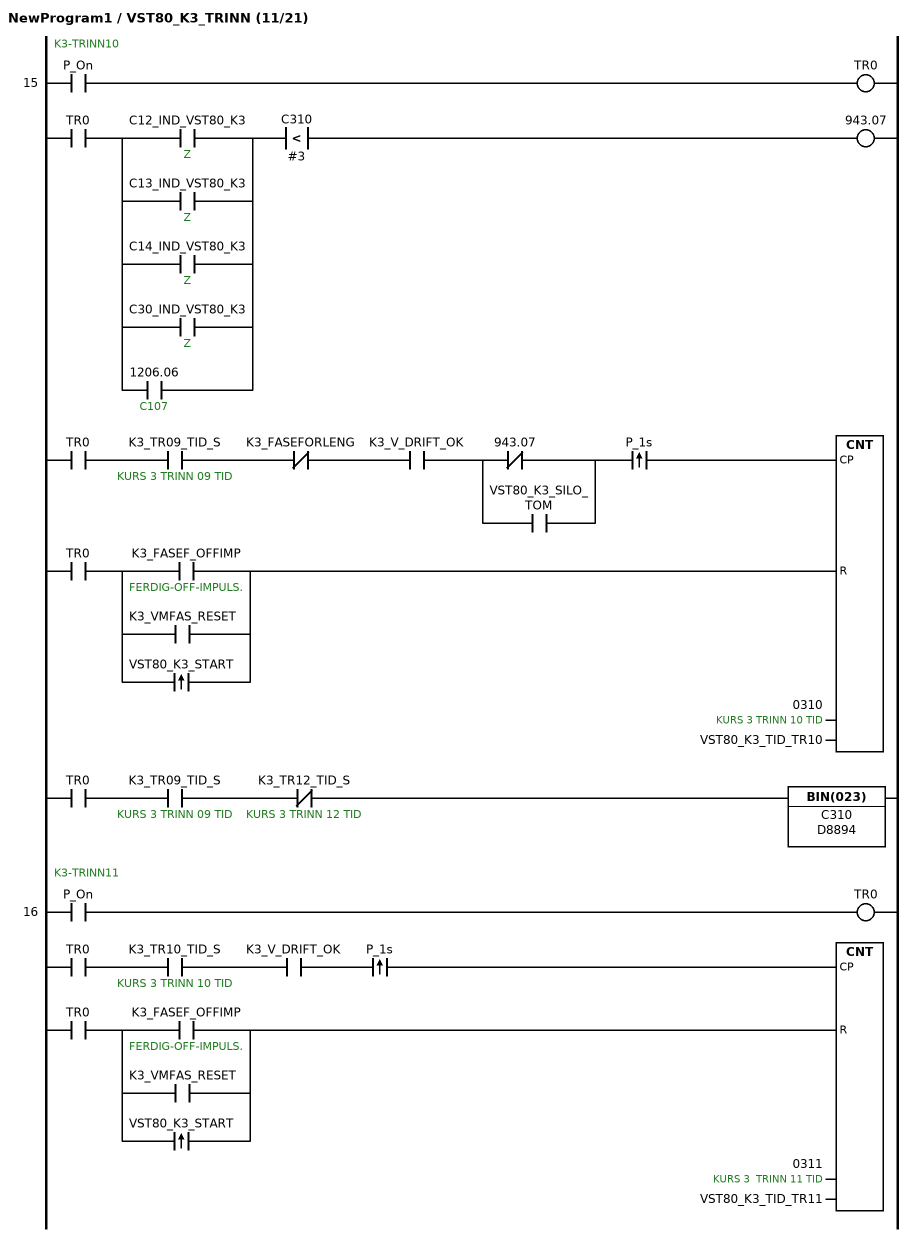
; rung 15: K3-TRINN10
LD P_On
OUT TR0
LD C12_IND_VST80_K3  ; Z
OR C13_IND_VST80_K3  ; Z
OR C14_IND_VST80_K3  ; Z
OR C30_IND_VST80_K3  ; Z
OR 1206.06  ; C107
ANDLD
AND<(310) C310 #3
OUT 943.07
LD TR0
AND K3_TR09_TID_S  ; KURS 3 TRINN 09 TID
ANDNOT K3_FASEFORLENG
AND K3_V_DRIFT_OK
LDNOT 943.07
OR VST80_K3_SILO_TOM
ANDLD
@AND P_1s
LD TR0
LD K3_FASEF_OFFIMP  ; FERDIG-OFF-IMPULS.
OR K3_VMFAS_RESET
@OR VST80_K3_START
ANDLD
CNT 0310 VST80_K3_TID_TR10  ; KURS 3 TRINN 10 TID
LD TR0
AND K3_TR09_TID_S  ; KURS 3 TRINN 09 TID
ANDNOT K3_TR12_TID_S  ; KURS 3 TRINN 12 TID
BIN(023) C310 D8894
; rung 16: K3-TRINN11
LD P_On
OUT TR0
AND K3_TR10_TID_S  ; KURS 3 TRINN 10 TID
AND K3_V_DRIFT_OK
@AND P_1s
LD TR0
LD K3_FASEF_OFFIMP  ; FERDIG-OFF-IMPULS.
OR K3_VMFAS_RESET
@OR VST80_K3_START
ANDLD
CNT 0311 VST80_K3_TID_TR11  ; KURS 3  TRINN 11 TID

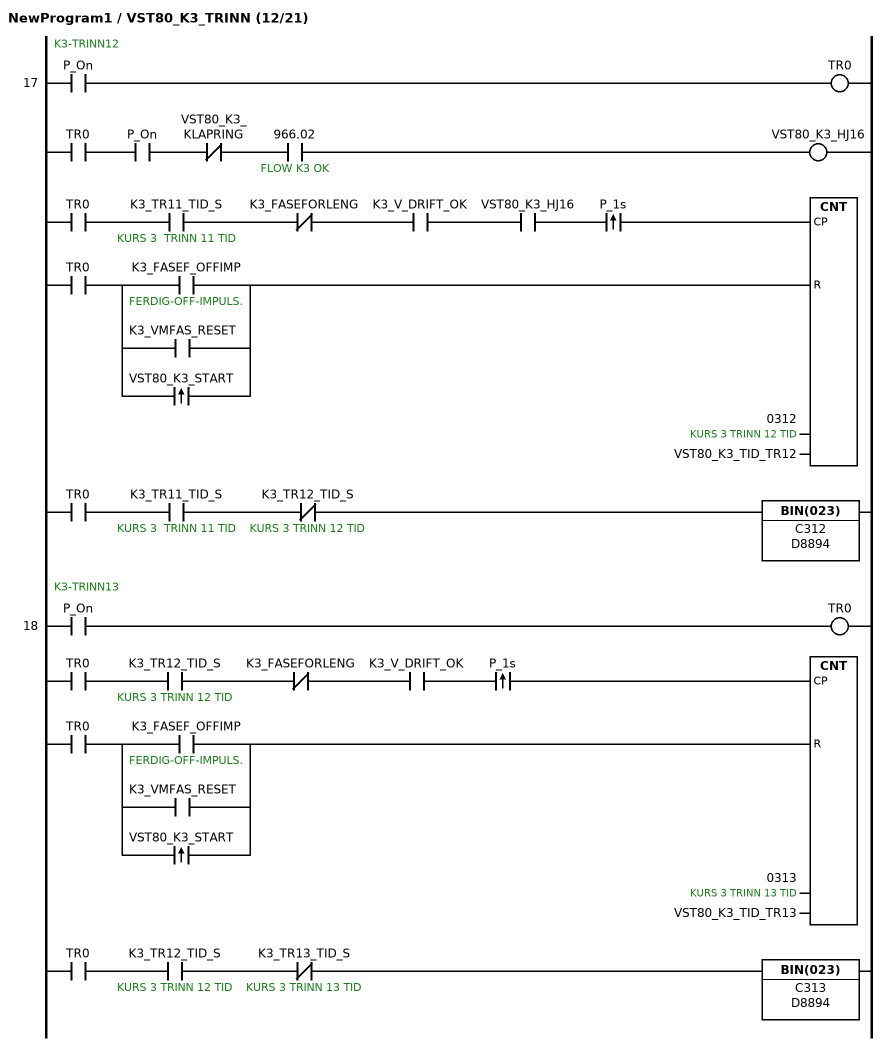
; rung 17: K3-TRINN12
LD P_On
OUT TR0
AND P_On
ANDNOT VST80_K3_KLAPRING
AND 966.02  ; FLOW K3 OK
OUT VST80_K3_HJ16
LD TR0
AND K3_TR11_TID_S  ; KURS 3  TRINN 11 TID
ANDNOT K3_FASEFORLENG
AND K3_V_DRIFT_OK
AND VST80_K3_HJ16
@AND P_1s
LD TR0
LD K3_FASEF_OFFIMP  ; FERDIG-OFF-IMPULS.
OR K3_VMFAS_RESET
@OR VST80_K3_START
ANDLD
CNT 0312 VST80_K3_TID_TR12  ; KURS 3 TRINN 12 TID
LD TR0
AND K3_TR11_TID_S  ; KURS 3  TRINN 11 TID
ANDNOT K3_TR12_TID_S  ; KURS 3 TRINN 12 TID
BIN(023) C312 D8894
; rung 18: K3-TRINN13
LD P_On
OUT TR0
AND K3_TR12_TID_S  ; KURS 3 TRINN 12 TID
ANDNOT K3_FASEFORLENG
AND K3_V_DRIFT_OK
@AND P_1s
LD TR0
LD K3_FASEF_OFFIMP  ; FERDIG-OFF-IMPULS.
OR K3_VMFAS_RESET
@OR VST80_K3_START
ANDLD
CNT 0313 VST80_K3_TID_TR13  ; KURS 3 TRINN 13 TID
LD TR0
AND K3_TR12_TID_S  ; KURS 3 TRINN 12 TID
ANDNOT K3_TR13_TID_S  ; KURS 3 TRINN 13 TID
BIN(023) C313 D8894

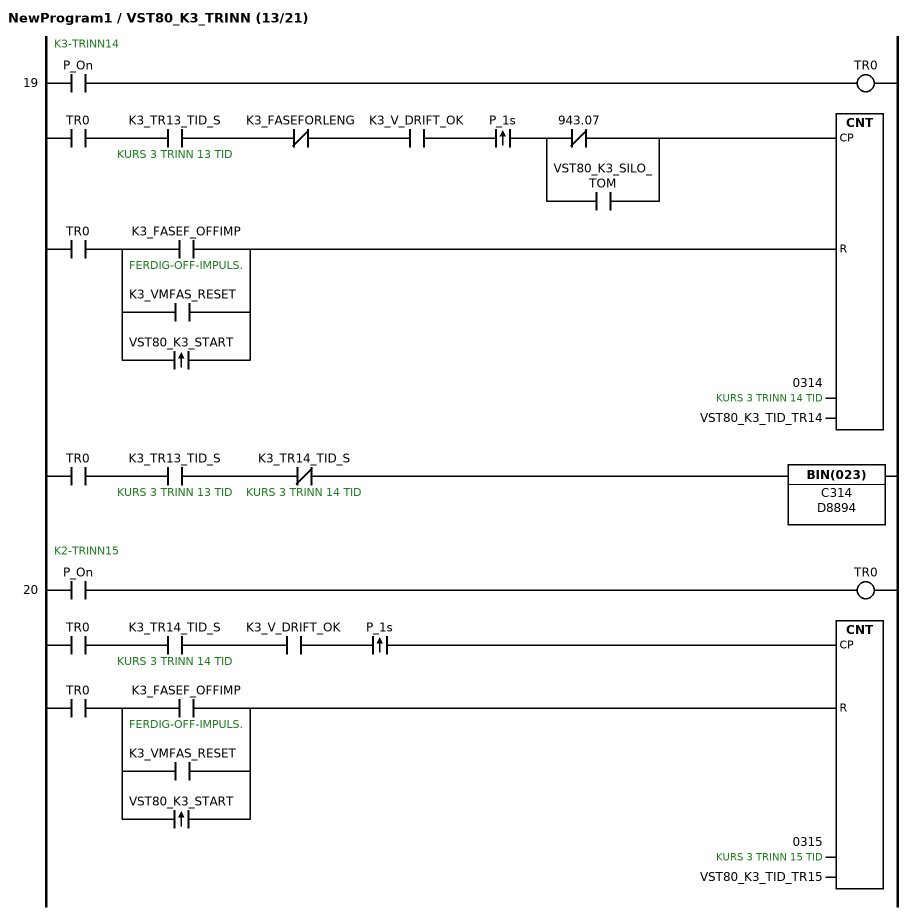
; rung 19: K3-TRINN14
LD P_On
OUT TR0
AND K3_TR13_TID_S  ; KURS 3 TRINN 13 TID
ANDNOT K3_FASEFORLENG
AND K3_V_DRIFT_OK
@AND P_1s
LDNOT 943.07
OR VST80_K3_SILO_TOM
ANDLD
LD TR0
LD K3_FASEF_OFFIMP  ; FERDIG-OFF-IMPULS.
OR K3_VMFAS_RESET
@OR VST80_K3_START
ANDLD
CNT 0314 VST80_K3_TID_TR14  ; KURS 3 TRINN 14 TID
LD TR0
AND K3_TR13_TID_S  ; KURS 3 TRINN 13 TID
ANDNOT K3_TR14_TID_S  ; KURS 3 TRINN 14 TID
BIN(023) C314 D8894
; rung 20: K2-TRINN15
LD P_On
OUT TR0
AND K3_TR14_TID_S  ; KURS 3 TRINN 14 TID
AND K3_V_DRIFT_OK
@AND P_1s
LD TR0
LD K3_FASEF_OFFIMP  ; FERDIG-OFF-IMPULS.
OR K3_VMFAS_RESET
@OR VST80_K3_START
ANDLD
CNT 0315 VST80_K3_TID_TR15  ; KURS 3 TRINN 15 TID

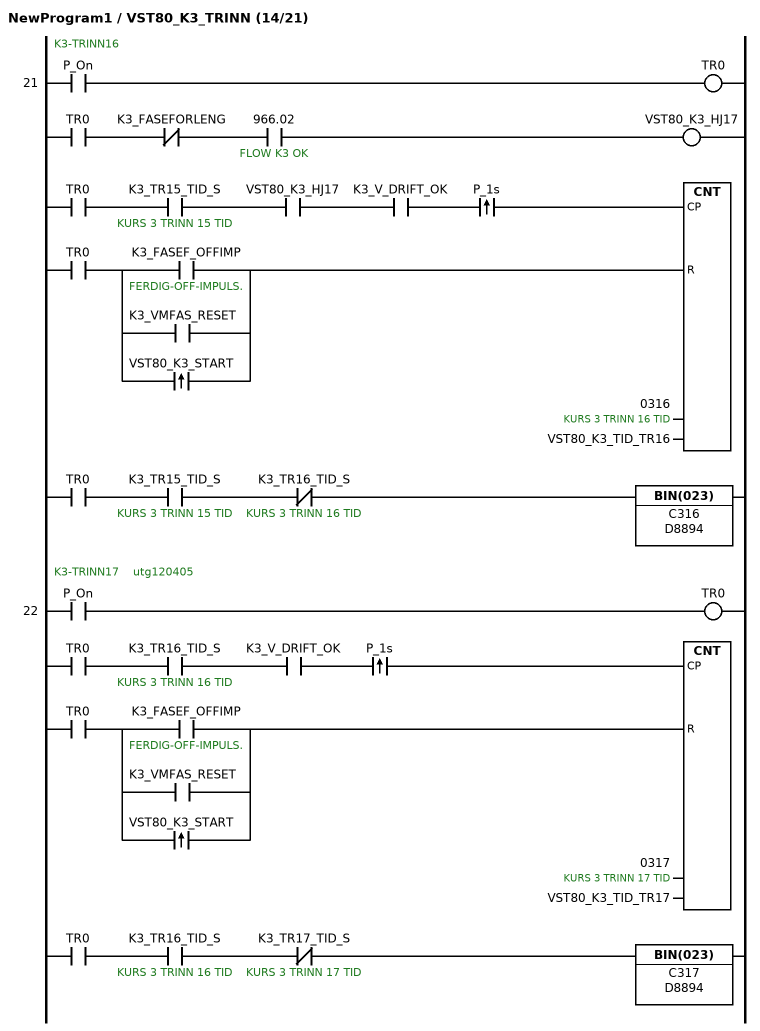
; rung 21: K3-TRINN16
LD P_On
OUT TR0
ANDNOT K3_FASEFORLENG
AND 966.02  ; FLOW K3 OK
OUT VST80_K3_HJ17
LD TR0
AND K3_TR15_TID_S  ; KURS 3 TRINN 15 TID
AND VST80_K3_HJ17
AND K3_V_DRIFT_OK
@AND P_1s
LD TR0
LD K3_FASEF_OFFIMP  ; FERDIG-OFF-IMPULS.
OR K3_VMFAS_RESET
@OR VST80_K3_START
ANDLD
CNT 0316 VST80_K3_TID_TR16  ; KURS 3 TRINN 16 TID
LD TR0
AND K3_TR15_TID_S  ; KURS 3 TRINN 15 TID
ANDNOT K3_TR16_TID_S  ; KURS 3 TRINN 16 TID
BIN(023) C316 D8894
; rung 22: K3-TRINN17    utg120405
LD P_On
OUT TR0
AND K3_TR16_TID_S  ; KURS 3 TRINN 16 TID
AND K3_V_DRIFT_OK
@AND P_1s
LD TR0
LD K3_FASEF_OFFIMP  ; FERDIG-OFF-IMPULS.
OR K3_VMFAS_RESET
@OR VST80_K3_START
ANDLD
CNT 0317 VST80_K3_TID_TR17  ; KURS 3 TRINN 17 TID
LD TR0
AND K3_TR16_TID_S  ; KURS 3 TRINN 16 TID
ANDNOT K3_TR17_TID_S  ; KURS 3 TRINN 17 TID
BIN(023) C317 D8894

